// TIA Portal V16 export
// export: Created 2022-02-02T12:03:29.6886658Z, ExportSetting WithDefaults, DisplayName Totally Integrated Automation Portal, DisplayVersion V16 Update 3, DisplayName TIA Portal Version Control Interface, DisplayVersion V16 Update 2, DisplayName TIA Portal Openness, DisplayVersion V16 Update 3, DisplayName STEP 7 Professional, DisplayVersion V16 Update 3, DisplayName STEP 7 Safety, DisplayVersion V16, DisplayName WinCC Professional, DisplayVersion V16 Update 3
TYPE "UT39512_Dy_DebugInst2Order"
TITLE = Dynamic UDT [Debug] — Second Order Response Simulation
// Second Order Response Simulation
// stored: IsFailsafeCompliant false
   STRUCT
      revInfo { ExternalWritable := 'False'} : "UT01000_St_SysRevision";   // ▀▀▀▀ UDT CURRENT REVISION
      ___________0010_0 { ExternalAccessible := 'False'; ExternalVisible := 'False'; ExternalWritable := 'False'} : Int;
      ___________0010_1 { ExternalAccessible := 'False'; ExternalVisible := 'False'; ExternalWritable := 'False'} : Int;   // ▀▀▀▀ CALCULATION CONSTANTS
      k_Gain : Real;   // CONSTANT — Simulation system gain
      k_NatFreq : Real;   // CONSTANT — Simulation natural frequency (rad/s)
      k_DampFactor : Real;   // CONSTANT — Simulation damping factor
      ___________0020_0 { ExternalAccessible := 'False'; ExternalVisible := 'False'; ExternalWritable := 'False'} : Int;
      ___________0020_1 { ExternalAccessible := 'False'; ExternalVisible := 'False'; ExternalWritable := 'False'} : Int;   // ▀▀▀▀ SIMULATION STATUS SIGNALS
      status_Running : Bool;   // STATUS — Simulation is running (1 = running, 0 = stopped)
      status_Stopped : Bool;   // STATUS — Simulation is stopped (not running) (1 = stopped, 0 = running)
      status_Stable : Bool;   // STATUS — Simulation response type is stable (1 = stable, 0 = unstable)
      status_OverDamp : Bool;   // STATUS — Response is stable/over damped (1 = stable, over damped)
      status_CritDamp : Bool;   // STATUS — Response is stable/critically damped (1 = stable, critically damped)
      status_UnderDamp : Bool;   // STATUS — Response is stable/under damped (1 = stable, under damped)
      status_Undamped : Bool;   // STATUS — Response is stable/undamped (1 = stable, undamped)
      status_USUnder : Bool;   // STATUS — Response is unstable/under damped (1 = unstable, under damped)
      status_USOver : Bool;   // STATUS — Response is unstable/over damped (1 = unstable, over damped)
      status_SteadyState : Bool;   // STATUS — Steady state (±2%) achieved (1 = In steady state, 0 = not steady state)
      status_Osc : Bool;   // STATUS — Oscillatory response (1 = oscillating response, 0 = non-oscillating)
      status_OscFreqRS : Real;   // STATUS — Frequency of oscillation, zero if non oscillatory (rad/s)
      status_OscFreqHz : Real;   // STATUS — Frequency of oscillation, zero if non oscillatory (Hz)
      status_Period : Real;   // STATUS — Period of oscillation, zero if non oscillatory (s)
      status_Aut : Bool;   // STATUS — Simulation is in automatic mode (1 = automatic, 0 = manual)
      status_Man : Bool;   // STATUS — Simulation is in manual mode (1 = manual, 0 = automatic)
      ___________0030_0 { ExternalAccessible := 'False'; ExternalVisible := 'False'; ExternalWritable := 'False'} : Int;
      ___________0030_1 { ExternalAccessible := 'False'; ExternalVisible := 'False'; ExternalWritable := 'False'} : Int;   // ▀▀▀▀ CALCULATED VALUES
      cal_PeakValue : Real;   // CALC — Peak output value
      cal_NatPeriod : Real;   // CALC — Period of natural oscillations (s)
      cal_DampFreq : Real;   // CALC — Damped frequency of the system (rad/s)
      cal_DampFreqHz : Real;   // CALC — Damped frequency of the system (Hz)
      cal_DampPeriod : Real;   // CALC — Period of damped oscillations (s)
      cal_TimeSteady : Real;   // CALC — Time to reach steady state, zero for unstable response (s)
      "cal_Time63%" : Real;   // CALC — Time to reach 63% of steady state (s)
      cal_TimePeak : Real;   // CALC — Time to reach the peak output value (s)
      ___________0040_0 { ExternalAccessible := 'False'; ExternalVisible := 'False'; ExternalWritable := 'False'} : Int;
      ___________0040_1 { ExternalAccessible := 'False'; ExternalVisible := 'False'; ExternalWritable := 'False'} : Int;   // ▀▀▀▀ OPERATING MODE SELECTION
      mode_AutMan : Bool;   // MODE — Automatic/manual mode selection (1 = auto mode, 0 = manual mode)
      mode_ManTime : Real;   // MODE — Manual mode time value (s)
      ___________0050_0 { ExternalAccessible := 'False'; ExternalVisible := 'False'; ExternalWritable := 'False'} : Int;
      ___________0050_1 { ExternalAccessible := 'False'; ExternalVisible := 'False'; ExternalWritable := 'False'} : Int;   // ▀▀▀▀ LIVE TIMING DATA
      actual_Output : Real;   // ACTUAL — SIMULATION OUTPUT VALUE (identical to OUTPUT parameter)
      actual_StartTime : DTL;   // ACTUAL — CPU time when simulation started
      actual_RunTime : Real;   // ACTUAL — Elapsed time since the simulation started (s)
   END_STRUCT;
   // revInfo.REV_BLOCK := 'UT39512';
   // revInfo.REV_NUMBER := '000.102';
   // revInfo.REV_DATE := '2022-02-02';
   // revInfo.REV_AUTHOR := 'M. Gledhill';
END_TYPE
